Staubli VAL3: stopMotor.pgx

program stopMotor()
begin
  stopMove()
  message="stopMotor:done"
  taskCreate "sendStatus",100,sendStatus()
  taskKill ("stopMotor")
end
